FUNCTION_BLOCK ARRAY2ARRAY_2_LREAL (* Service Interface Function Block Type *)
  (* Description: Copyright (c) 2014 Profactor GmbH This program and the accompanying materials are made available under the terms of the Eclipse Public License 2.0 which is available at https://www.eclipse.org/legal/epl-2.0/ SPDX-License-Identifier: EPL-2.0 *)
  (* Version 3.0, 2025-04-14, Patrick Aigner, changed package *)
  (* Version 1.0, 2014-08-05, Matthias Plasch, Profactor GmbH *)
  PACKAGE eclipse4diac::convert;
  {SET_ATTRIBUTE(eclipse4diac::core::GenericClassName, 'GEN_ARRAY2ARRAY')}
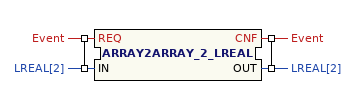
  EVENT_INPUT
    REQ WITH IN; (* Service Request *)
  END_EVENT
  EVENT_OUTPUT
    CNF WITH OUT; (* Confirmation of Requested Service *)
  END_EVENT
  VAR_INPUT
    IN : ARRAY [0..1] OF LREAL; (* array input *)
  END_VAR
  VAR_OUTPUT
    OUT : ARRAY [0..1] OF LREAL; (* array output *)
  END_VAR
END_FUNCTION_BLOCK
